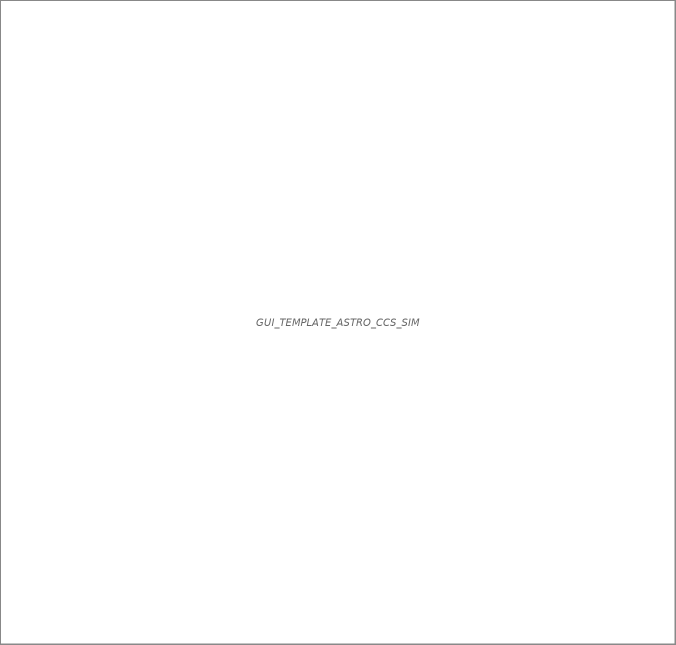
VISUALIZATION GUI_ASTRO_CCS_SIM  // 676x645
    Frame (0,0 676x645)
        shows GUI_TEMPLATE_ASTRO_CCS_SIM(m_DeviceName := 'astro', m_Instance := MAIN.astro)
END_VISUALIZATION

(* stored: Version 1.1.0.1, ProductVersion 3.1.4024.12
   Visu GUI_ASTRO_CCS_SIM: Id {b56db7a4-8ee3-4993-9130-35151cd4f7eb} *)
